(* CODESYS project CRTL_QUALD.project

Project tree, tasks and I/O mapping:
  Device : CODESYS Control Win V3, 3S - Smart Software Solutions GmbH, order no. 305021, version 3.5.11.30
    application Application
      libraries: Standard, * (System)
      task MainTask (cyclic, interval t#20ms, priority 1) calls PLC_PRG
      task VISU_TASK (cyclic, interval 100 ms, priority 31) calls VisuElems.Visu_Prg
      program PLC_PRG [LD]
      visualisation Visualization
  libraries: VisuSymbols, 3.5.10.0 (System)
  text list GlobalTextList
*)

// Device/Application/PLC_PRG
PROGRAM PLC_PRG
VAR
	EST1             : BOOL;
    SENSOR_SUCO      : BOOL;
    PNEUMATICO       : BOOL;
    EST2             : BOOL;
    ALARME           : BOOL;
    DESLIGA_ESTEIRA  : BOOL;
	START            : BOOL;
	STOP             : BOOL;
	P1               : BOOL;
	P2               : BOOL;
	P3: BOOL;
	TOF_1: TOF;
	ET1: TIME;
	P4: BOOL;
	AUX: BOOL;
END_VAR
VAR // added by the converter: edge detectors and wires of the graphical bodies
    _w1 : BOOL;
    _ft1 : F_TRIG;
END_VAR

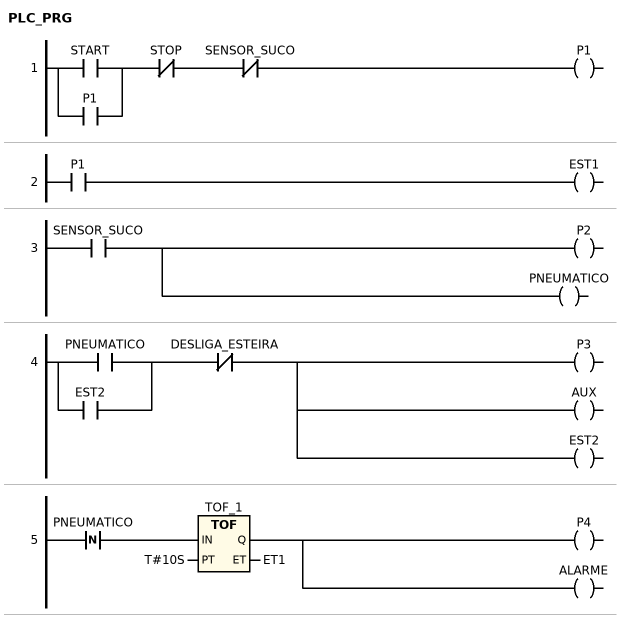
// NETWORK 1
P1 := (START OR P1) AND NOT STOP AND NOT SENSOR_SUCO;

// NETWORK 2
EST1 := P1;

// NETWORK 3
P2 := SENSOR_SUCO;
PNEUMATICO := SENSOR_SUCO;

// NETWORK 4
_w1 := (PNEUMATICO OR EST2) AND NOT DESLIGA_ESTEIRA;
P3 := _w1;
AUX := _w1;
EST2 := _w1;

// NETWORK 5
_ft1(CLK := PNEUMATICO);
TOF_1(IN := _ft1.Q, PT := T#10S, ET => ET1); // TOF
P4 := TOF_1.Q;
ALARME := TOF_1.Q;

END_PROGRAM

// Device/Application/Visualization
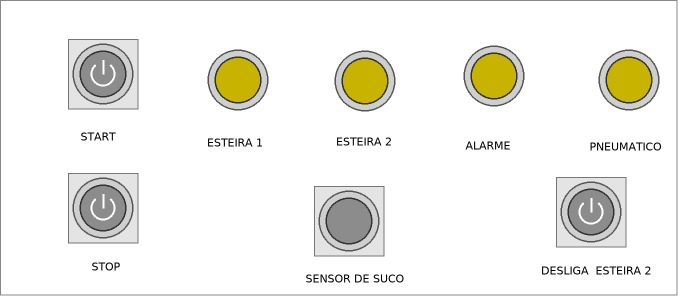
VISUALIZATION Visualization  // 678x296
    PowerSwitch (68,39 70x70), variable: PLC_PRG.START, behaviour: TAP, style: Switch-PowerSwitch-Gray
    Lamp1 (203,45 70x70), variable: PLC_PRG.EST1, style: Lamp-Lamp1-Yellow
    Lamp1 (330,46 70x70), variable: PLC_PRG.EST2, style: Lamp-Lamp1-Yellow
    Lamp1 (459,41 70x70), variable: PLC_PRG.ALARME, style: Lamp-Lamp1-Yellow
    Label (56,122 84x30), "START"
    PowerSwitch (68,173 70x70), variable: PLC_PRG.STOP, behaviour: TOGGLE, style: Switch-PowerSwitch-Gray
    Label (64,252 84x30), "STOP"
    Label (193,128 84x30), "ESTEIRA 1"
    Label (322,127 84x30), "ESTEIRA 2"
    Label (446,131 84x30), "ALARME"
    Label (293,264 124x30), "SENSOR DE SUCO"
    Lamp1 (594,45 70x70), variable: PLC_PRG.PNEUMATICO, style: Lamp-Lamp1-Yellow
    Label (575,132 101x30), "PNEUMATICO"
    PowerSwitch (556,177 70x70), variable: PLC_PRG.DESLIGA_ESTEIRA, behaviour: TOGGLE, style: Switch-PowerSwitch-Gray
    Label (526,256 141x30), "DESLIGA ESTEIRA 2"
    PushSwitchLed (314,186 70x70), variable: PLC_PRG.SENSOR_SUCO, behaviour: TOGGLE, style: Switch-PushSwitchLed-Gray
END_VISUALIZATION
